(*
Nazwa:			P02_BottlePusher
Opis:			Stacja wbijaka butelek
Wersja:			v0.1
Data:			2024-05-21
Autor:			DP
Urzadzenia:		
Konfiguracja:	
Info:
*)

PROGRAM P02_BottlePusher
VAR
	
	fbBottlePusher									:FB_Gate;
	eBottlePusherState								:E_Station; 									
	eBottlePusherRunningState						:E_Barrier; 
	fbBottlePusherState								:FB_State;	

	QbBottlePusherActuator 							:BOOL;
	IbBottlePusherActuatorSensor 			AT %I*  :BOOL; 
	IbBottlePusherBottleBeforeSensor 		AT %I*  :BOOL; 
	IbBottlePusherBottleAfterSensor 		AT %I*  :BOOL;

	
	tonfbBottlePusherDownSensor						:TON;
END_VAR

aBottlePusher();


tonfbBottlePusherDownSensor	(IN:= QbBottlePusherActuator, PT:=T#500MS);

ACTION aBottlePusher:
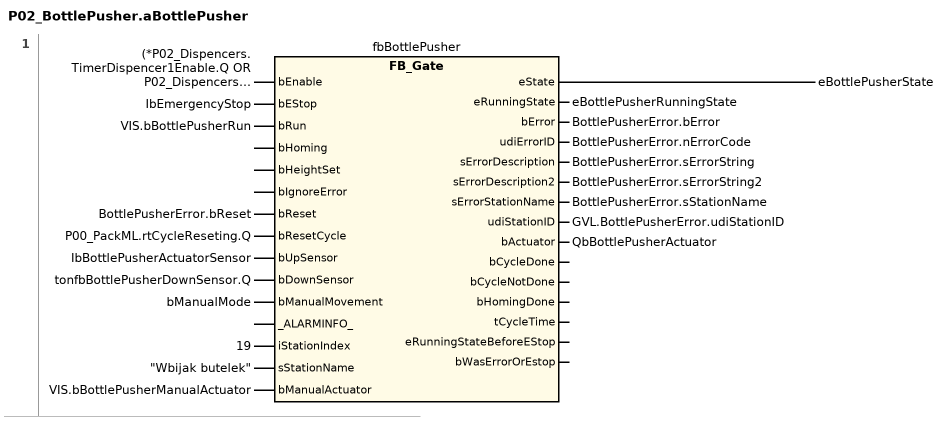
// NETWORK 1
fbBottlePusher(
    bEnable := (*P02_Dispencers.TimerDispencer1Enable.Q OR P02_Dispencers.TimerDispencer3Enable.Q*)FALSE,
    bEStop := IbEmergencyStop,
    bRun := VIS.bBottlePusherRun,
    bReset := BottlePusherError.bReset,
    bResetCycle := P00_PackML.rtCycleReseting.Q,
    bUpSensor := IbBottlePusherActuatorSensor,
    bDownSensor := tonfbBottlePusherDownSensor.Q,
    bManualMovement := bManualMode,
    iStationIndex := 19,
    sStationName := "Wbijak butelek",
    bManualActuator := VIS.bBottlePusherManualActuator,
    eRunningState => eBottlePusherRunningState,
    bError => BottlePusherError.bError,
    udiErrorID => BottlePusherError.nErrorCode,
    sErrorDescription => BottlePusherError.sErrorString,
    sErrorDescription2 => BottlePusherError.sErrorString2,
    sErrorStationName => BottlePusherError.sStationName,
    udiStationID => GVL.BottlePusherError.udiStationID,
    bActuator => QbBottlePusherActuator); // FB_Gate
eBottlePusherState := fbBottlePusher.eState;
END_ACTION

END_PROGRAM

(* stored: Version 1.1.0.1, ProductVersion 3.1.4026.13, FileIdentifier d88f566b1189c3bdb504ff19c47e70c213685739, FileSignature 0f672405432b065a15c4eff3c133492ae68ea24f97a371b606a6a9eb6496199cb20adeff8ac24ba93f3bf6202de8ae28fc1d05671ccf593e6cc73a446a2514eec10b55ac7b6ac8dc0fe8661427ee87bb17870145bbd0a1f4b90e8339937120562103eb04973727c8e7d37ec915de1b75e14f519451abdd76b47850220418d70e99e909bbf16ea5178cd1ee1330596da2934e3a0f383c87b2d49f8e164bdf19f02d03d70475d1e5eaa57196c4e4ccea0fbc59bd13b11ecaa0022b334f706fa31d062ebe48c486eb251abbee05f5e1923554e4dbdd90ccc7040a662fdbe6109ef71d5fc5c76d123e28f30bf88259c8fa59a2d0de7680c50417bfd219a5a8aafe6b
   POU P02_BottlePusher: Id {fb88f823-744f-4661-a624-b68e8d941d4b}, SpecialFunc None
   Action aBottlePusher: Id {1d48e357-bccd-43f3-bb62-b493ad2b3f51} *)
